// TIA Portal project "MetalCuttingLine" (V17)
// End to End

(* hardware
DEVICE "S7-1500/ET200MP station_1"  S7-1500 station
   slot 0: "Rail_0"  Rack  6ES7 590-1***0-0AA0
   slot 1: "PLC_1"  CPU 1516-3 PN/DP  6ES7 516-3AN02-0AB0  V2.9
      slot 3: "CPU display_1"  6ES7591-1BA00-0AA0
      slot 32768: "PROFINET interface_1"  X1
         slot 32769: "Port_1"  X1 P1
         slot 32770: "Port_2"  X1 P2
      slot 33024: "PROFINET interface_2"  X2
         slot 33025: "Port_1"  X2 P1
      slot 33280: "DP interface_1"  X3
      slot 34817: "Virtual CP interface port_1"  Virtual CP interface port  Virtual CP interface port
DEVICE "HMI_1"  KTP900 Basic PN
   slot 0: "HMI_1"  KTP900 Basic PN  6AV2 123-2JB03-0AX0  17.0.0.0
   slot 1: "HMI_RT_1"  KTP900 Basic PN  6AV2 123-2JB03-0AX0  17.0.0.0
   slot 5: "HMI_1.IE_CP_1"  PROFINET Interface  17.0.0.0
      slot 1: "PROFINET Interface_1"  PROFINET Interface
         slot 1: "Port_1"  Port
*)

// ===== PLC "PLC_1"  CPU 1516-3 PN/DP =====

VAR_GLOBAL   // PLC tag table "IO_Tags"
   "I_StartPB" AT %I0.0 : Bool;   // Start pushbutton
   "I_StopPB" AT %I0.1 : Bool;   // Stop pushbutton
   "I_EStop" AT %I0.2 : Bool;   // Emergency stop (NC contact)
   "I_AutoManSwitch" AT %I0.3 : Bool;   // Mode select switch
   "I_ClampRetracted" AT %I0.4 : Bool;   // Clamp cylinder retracted limit switch
   "I_ClampExtended" AT %I0.5 : Bool;   // Clamp cylinder extended limit switch
   "I_ShearRetracted" AT %I0.6 : Bool;   // Shear cylinder retracted limit switch
   "I_ShearExtended" AT %I0.7 : Bool;   // Shear cylinder extended limit switch
   "I_PartAtEject" AT %I1.0 : Bool;   // Photoeye at eject station
   "Q_FeedMotor" AT %Q0.0 : Bool;   // Feed conveyor motor run
   "Q_ClampExtend" AT %Q0.1 : Bool;   // Clamp cylinder extend solenoid
   "Q_ClampRetract" AT %Q0.2 : Bool;   // Clamp cylinder retract solenoid
   "Q_ShearExtend" AT %Q0.3 : Bool;   // Shear cylinder extend solenoid
   "Q_ShearRetract" AT %Q0.4 : Bool;   // Shear cylinder retract solenoid
   "Q_EjectGoodLane" AT %Q0.5 : Bool;   // Diverter to good-parts lane
   "Q_EjectScrapLane" AT %Q0.6 : Bool;   // Diverter to scrap lane
   "Q_RunLamp" AT %Q0.7 : Bool;   // Auto-run indicator lamp
   "Q_FaultLamp" AT %Q1.0 : Bool;   // Fault/alarm indicator lamp
END_VAR

DATA_BLOCK "Recipe_Status"   // DB1
{ S7_Optimized_Access := 'FALSE' }
VERSION : 0.1
   VAR
      Recipe : Struct
         TargetLength : Real := 500.0;   // Target cut length in mm
         Tolerance : Real := 2.0;   // Allowed+- tolerance in mm
         FeedSpeed : Real := 50.0;   // Feed Conveyor speed referenc %
      END_STRUCT;
      Status : Struct
         CurrentLength : Real := 0.0;   // Live measured length from the encoder
         GoodCount : Int;   // Total good pieces cut
         ScrapCount : Int;   // Total scrap pieces out
         TotalCount : Int;   // Total pieces cut (good+scrap)
      END_STRUCT;
      Mode : Struct
         AutoMode : Bool;   // True when in Auto mode
         ManualMode : Bool;   // True when in Manual mode
         Running : Bool;   // True when machine cycle is active
      END_STRUCT;
      Alarms : Struct
         EstopTripped : Bool;   // Emergency stop active
         ClampFault : Bool;   // Clamp cylinder failed to reach position
         ShearFault : Bool;   // Shear cylinder failed to reach position
         LengthError : Bool;   // Measured length out of expected range
         AnyFaultActive : Bool;   // True if any single fault active
         AlarmWord : Word;   // alarmWord
      END_STRUCT;
   END_VAR
BEGIN
END_DATA_BLOCK

DATA_BLOCK "ModeControl_DB"   // DB2
{ S7_Optimized_Access := 'TRUE' }
VERSION : 0.1
// stored: InstanceOfName ModeControl
"ModeControl"
BEGIN
END_DATA_BLOCK

DATA_BLOCK "FeedConveyor_DB"   // DB3
{ S7_Optimized_Access := 'TRUE' }
VERSION : 0.1
// stored: InstanceOfName FeedConveyor
"FeedConveyor"
BEGIN
END_DATA_BLOCK

DATA_BLOCK "LengthMeasurement_DB"   // DB4
{ S7_Optimized_Access := 'TRUE' }
VERSION : 0.1
// stored: InstanceOfName LengthMeasurement
"LengthMeasurement"
BEGIN
END_DATA_BLOCK

DATA_BLOCK "ShearCylinder_DB"   // DB5
{ S7_Optimized_Access := 'TRUE' }
VERSION : 0.1
// stored: InstanceOfName ShearCylinder
"ShearCylinder"
BEGIN
END_DATA_BLOCK

DATA_BLOCK "ClampCylinder_DB"   // DB6
{ S7_Optimized_Access := 'TRUE' }
VERSION : 0.1
// stored: InstanceOfName ClampCylinder
"ClampCylinder"
BEGIN
END_DATA_BLOCK

DATA_BLOCK "EjectSort_DB"   // DB7
{ S7_Optimized_Access := 'TRUE' }
VERSION : 0.1
// stored: InstanceOfName EjectSort
"EjectSort"
BEGIN
END_DATA_BLOCK

DATA_BLOCK "AlarmHandler_DB"   // DB8
{ S7_Optimized_Access := 'TRUE' }
VERSION : 0.1
// stored: InstanceOfName AlarmHandler
"AlarmHandler"
BEGIN
END_DATA_BLOCK

FUNCTION_BLOCK "ModeControl"   // FB1, LAD
{ S7_Optimized_Access := 'TRUE' }
VERSION : 0.1
   VAR_INPUT
      StartPB : Bool;
      StopPB : Bool;
      EStop : Bool;
      AutManSwitch : Bool;
   END_VAR
BEGIN

REGION Network 1: Start/Stop seal in Rung
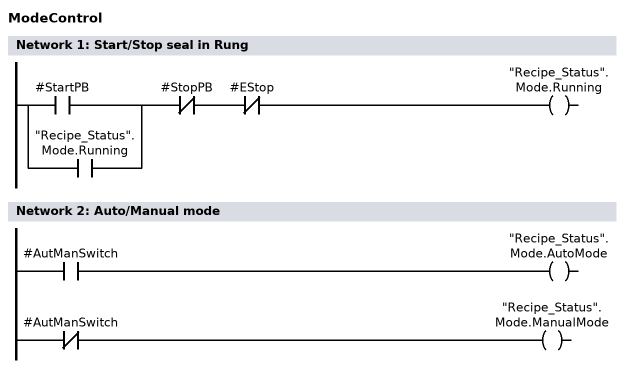
   RUNG wire#powerrail
      Contact( #StartPB )
      wire#w1
      I_Contact( #StopPB )
      I_Contact( #EStop )
      Coil( "Recipe_Status".Mode.Running )
   END_RUNG
   RUNG wire#powerrail
      Contact( "Recipe_Status".Mode.Running )
   END_RUNG wire#w1
   // the same network as SCL:
   "Recipe_Status".Mode.Running := (#StartPB OR "Recipe_Status".Mode.Running) AND NOT #StopPB AND NOT #EStop;
END_REGION

REGION Network 2: Auto/Manual mode
   RUNG wire#powerrail
      Contact( #AutManSwitch )
      Coil( "Recipe_Status".Mode.AutoMode )
   END_RUNG
   RUNG wire#powerrail
      I_Contact( #AutManSwitch )
      Coil( "Recipe_Status".Mode.ManualMode )
   END_RUNG
   // the same network as SCL:
   "Recipe_Status".Mode.AutoMode := #AutManSwitch;
   "Recipe_Status".Mode.ManualMode := NOT #AutManSwitch;
END_REGION
END_FUNCTION_BLOCK

FUNCTION_BLOCK "FeedConveyor"   // FB2, LAD
{ S7_Optimized_Access := 'TRUE' }
VERSION : 0.1
   VAR_INPUT
      LengthReached : Bool;
   END_VAR
   VAR_IN_OUT
      FeedMotorOn : Bool;
   END_VAR
BEGIN

REGION Network 1
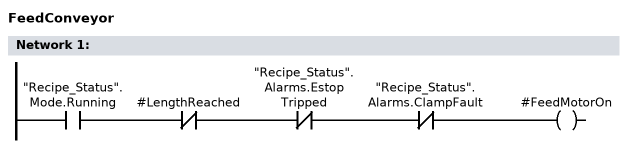
   RUNG wire#powerrail
      Contact( "Recipe_Status".Mode.Running )
      I_Contact( #LengthReached )
      I_Contact( "Recipe_Status".Alarms.EstopTripped )
      I_Contact( "Recipe_Status".Alarms.ClampFault )
      Coil( #FeedMotorOn )
   END_RUNG
   // the same network as SCL:
   #FeedMotorOn := "Recipe_Status".Mode.Running AND NOT #LengthReached AND NOT "Recipe_Status".Alarms.EstopTripped AND NOT "Recipe_Status".Alarms.ClampFault;
END_REGION
END_FUNCTION_BLOCK

FUNCTION_BLOCK "LengthMeasurement"   // FB3, LAD
{ S7_Optimized_Access := 'TRUE' }
VERSION : 0.1
   VAR_INPUT
      FeedMotorOn : Bool;
      ResetRamp : Bool;
   END_VAR
   VAR_OUTPUT
      LengthReached : Bool;
   END_VAR
   VAR
      RampAccum : Real;
      ToleranceCheck : Real;
   END_VAR
BEGIN

REGION Network 1: Accumulate Simulated Length
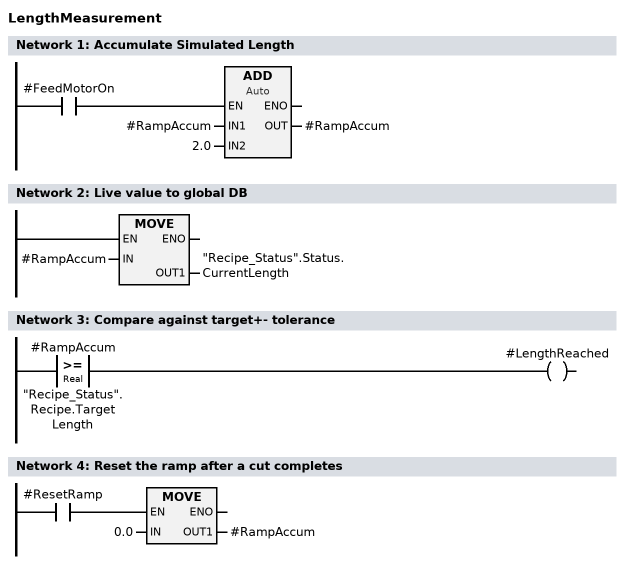
   RUNG wire#powerrail
      Contact( #FeedMotorOn )
      Add(in1 := #RampAccum, in2 := 2.0, out => #RampAccum)
   END_RUNG
   // the same network as SCL:
   IF #FeedMotorOn THEN #RampAccum := #RampAccum + 2.0; END_IF;
END_REGION

REGION Network 2: Live value to global DB
   RUNG wire#powerrail
      Move(in := #RampAccum, out1 => "Recipe_Status".Status.CurrentLength)
   END_RUNG
   // the same network as SCL:
   "Recipe_Status".Status.CurrentLength := #RampAccum;
END_REGION

REGION Network 3: Compare against target+- tolerance
   RUNG wire#powerrail
      { S7_Templates := "SrcType := Real" } GE_Contact(in1 := #RampAccum, in2 := "Recipe_Status".Recipe.TargetLength)
      Coil( #LengthReached )
   END_RUNG
   // the same network as SCL:
   #LengthReached := #RampAccum >= "Recipe_Status".Recipe.TargetLength;
END_REGION

REGION Network 4: Reset the ramp after a cut completes
   RUNG wire#powerrail
      Contact( #ResetRamp )
      Move(in := 0.0, out1 => #RampAccum)
   END_RUNG
   // the same network as SCL:
   IF #ResetRamp THEN #RampAccum := 0.0; END_IF;
END_REGION
END_FUNCTION_BLOCK

FUNCTION_BLOCK "ClampCylinder"   // FB4, LAD
{ S7_Optimized_Access := 'TRUE' }
VERSION : 0.1
   VAR_INPUT
      StartClamp : Bool;
      RetractClamp : Bool;
      ClampRetractedSensor : Bool;
      ClampExtendedSensor : Bool;
   END_VAR
   VAR_OUTPUT
      ClampExtendedCoil : Bool;
      ClampRetractCoil : Bool;
      ClampInPosition : Bool;
   END_VAR
   VAR
      "Step" : Int;
   END_VAR
   VAR_TEMP   // added for the SCL form of the ladder/FBD networks
      _w1 : Bool;
   END_VAR
BEGIN

REGION Network 1: Step0--> Step1 (Start Extending)
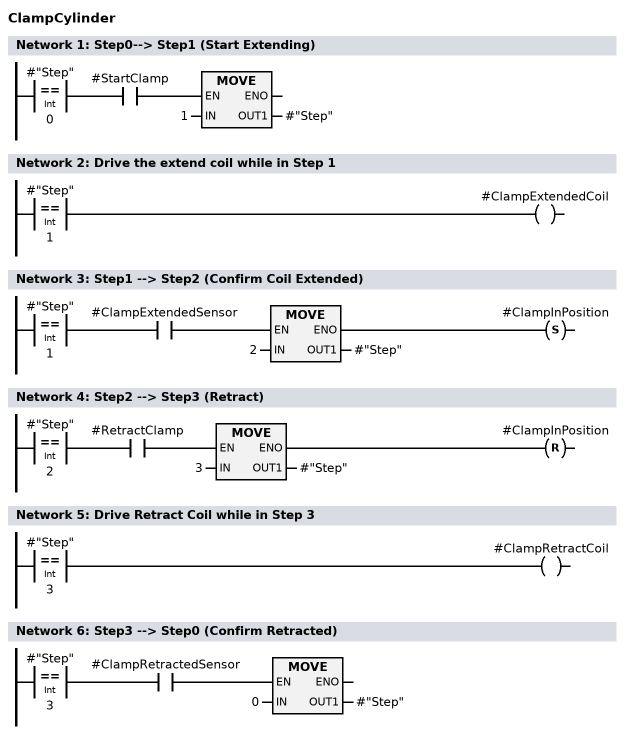
   RUNG wire#powerrail
      { S7_Templates := "SrcType := Int" } EQ_Contact(in1 := #"Step", in2 := 0)
      Contact( #StartClamp )
      Move(in := 1, out1 => #"Step")
   END_RUNG
   // the same network as SCL:
   IF (#"Step" = 0) AND #StartClamp THEN #"Step" := 1; END_IF;
END_REGION

REGION Network 2: Drive the extend coil while in Step 1
   RUNG wire#powerrail
      { S7_Templates := "SrcType := Int" } EQ_Contact(in1 := #"Step", in2 := 1)
      Coil( #ClampExtendedCoil )
   END_RUNG
   // the same network as SCL:
   #ClampExtendedCoil := #"Step" = 1;
END_REGION

REGION Network 3: Step1 --> Step2 (Confirm Coil Extended)
   RUNG wire#powerrail
      { S7_Templates := "SrcType := Int" } EQ_Contact(in1 := #"Step", in2 := 1)
      Contact( #ClampExtendedSensor )
      Move(in := 2, out1 => #"Step")
      S_Coil( #ClampInPosition )
   END_RUNG
   // the same network as SCL:
   #_w1 := (#"Step" = 1) AND #ClampExtendedSensor;
   IF #_w1 THEN
       #"Step" := 2;
       #ClampInPosition := TRUE;
   END_IF;
END_REGION

REGION Network 4: Step2 --> Step3 (Retract)
   RUNG wire#powerrail
      { S7_Templates := "SrcType := Int" } EQ_Contact(in1 := #"Step", in2 := 2)
      Contact( #RetractClamp )
      Move(in := 3, out1 => #"Step")
      R_Coil( #ClampInPosition )
   END_RUNG
   // the same network as SCL:
   #_w1 := (#"Step" = 2) AND #RetractClamp;
   IF #_w1 THEN
       #"Step" := 3;
       #ClampInPosition := FALSE;
   END_IF;
END_REGION

REGION Network 5: Drive Retract Coil while in Step 3
   RUNG wire#powerrail
      { S7_Templates := "SrcType := Int" } EQ_Contact(in1 := #"Step", in2 := 3)
      Coil( #ClampRetractCoil )
   END_RUNG
   // the same network as SCL:
   #ClampRetractCoil := #"Step" = 3;
END_REGION

REGION Network 6: Step3 --> Step0 (Confirm Retracted)
   RUNG wire#powerrail
      { S7_Templates := "SrcType := Int" } EQ_Contact(in1 := #"Step", in2 := 3)
      Contact( #ClampRetractedSensor )
      Move(in := 0, out1 => #"Step")
   END_RUNG
   // the same network as SCL:
   IF (#"Step" = 3) AND #ClampRetractedSensor THEN #"Step" := 0; END_IF;
END_REGION
END_FUNCTION_BLOCK

FUNCTION_BLOCK "ShearCylinder"   // FB5, LAD
{ S7_Optimized_Access := 'TRUE' }
VERSION : 0.1
   VAR_INPUT
      StartShear : Bool;
      ShearRetractedSensor : Bool;
      ShearExtendedSensor : Bool;
   END_VAR
   VAR_OUTPUT
      ShearExtendCoil : Bool;
      ShearRetractCoil : Bool;
      CutComplete : Bool;
   END_VAR
   VAR
      "Step" : Int;
      FaultTimer : IEC_TIMER;
   END_VAR
   VAR_TEMP   // added for the SCL form of the ladder/FBD networks
      _w1 : Bool;
   END_VAR
BEGIN

REGION Network 1: Start Extending
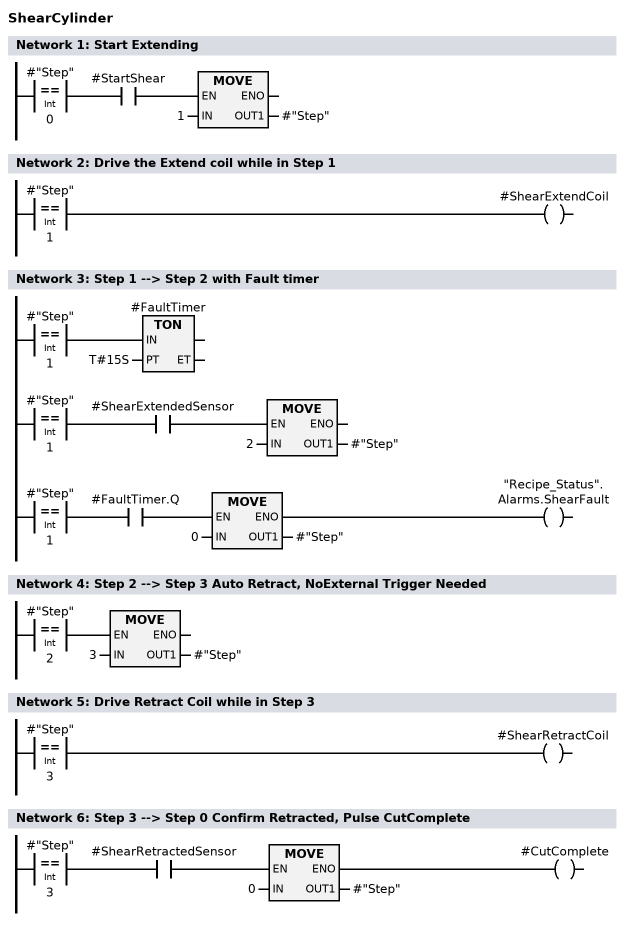
   RUNG wire#powerrail
      { S7_Templates := "SrcType := Int" } EQ_Contact(in1 := #"Step", in2 := 0)
      Contact( #StartShear )
      Move(in := 1, out1 => #"Step")
   END_RUNG
   // the same network as SCL:
   IF (#"Step" = 0) AND #StartShear THEN #"Step" := 1; END_IF;
END_REGION

REGION Network 2: Drive the Extend coil while in Step 1
   RUNG wire#powerrail
      { S7_Templates := "SrcType := Int" } EQ_Contact(in1 := #"Step", in2 := 1)
      Coil( #ShearExtendCoil )
   END_RUNG
   // the same network as SCL:
   #ShearExtendCoil := #"Step" = 1;
END_REGION

REGION Network 3: Step 1 --> Step 2 with Fault timer
   #FaultTimer.TON(IN := #"Step" = 1, PT := T#15S);
   IF (#"Step" = 1) AND #ShearExtendedSensor THEN #"Step" := 2; END_IF;
   #_w1 := (#"Step" = 1) AND #FaultTimer.Q;
   IF #_w1 THEN #"Step" := 0; END_IF;
   "Recipe_Status".Alarms.ShearFault := #_w1;
END_REGION

REGION Network 4: Step 2 --> Step 3 Auto Retract, NoExternal Trigger Needed
   RUNG wire#powerrail
      { S7_Templates := "SrcType := Int" } EQ_Contact(in1 := #"Step", in2 := 2)
      Move(in := 3, out1 => #"Step")
   END_RUNG
   // the same network as SCL:
   IF #"Step" = 2 THEN #"Step" := 3; END_IF;
END_REGION

REGION Network 5: Drive Retract Coil while in Step 3
   RUNG wire#powerrail
      { S7_Templates := "SrcType := Int" } EQ_Contact(in1 := #"Step", in2 := 3)
      Coil( #ShearRetractCoil )
   END_RUNG
   // the same network as SCL:
   #ShearRetractCoil := #"Step" = 3;
END_REGION

REGION Network 6: Step 3 --> Step 0 Confirm Retracted, Pulse CutComplete
   RUNG wire#powerrail
      { S7_Templates := "SrcType := Int" } EQ_Contact(in1 := #"Step", in2 := 3)
      Contact( #ShearRetractedSensor )
      Move(in := 0, out1 => #"Step")
      Coil( #CutComplete )
   END_RUNG
   // the same network as SCL:
   #_w1 := (#"Step" = 3) AND #ShearRetractedSensor;
   IF #_w1 THEN #"Step" := 0; END_IF;
   #CutComplete := #_w1;
END_REGION
END_FUNCTION_BLOCK

FUNCTION_BLOCK "EjectSort"   // FB6, LAD
{ S7_Optimized_Access := 'TRUE' }
VERSION : 0.1
   VAR_INPUT
      PartAtEject : Bool;
   END_VAR
   VAR_OUTPUT
      EjectGoodCoil : Bool;
      EjectScrapCoil : Bool;
   END_VAR
   VAR
      GoodEdgeMem : Bool;
      ScrapEdgeMem : Bool;
   END_VAR
   VAR_TEMP
      LengthDiff : Real;
      WithinTolerance : Bool;
   END_VAR
   VAR_TEMP   // added for the SCL form of the ladder/FBD networks
      _w1 : Bool;
      _w2 : Bool;
   END_VAR
BEGIN

REGION Network 1: Calculate whether the cut was within tolerance
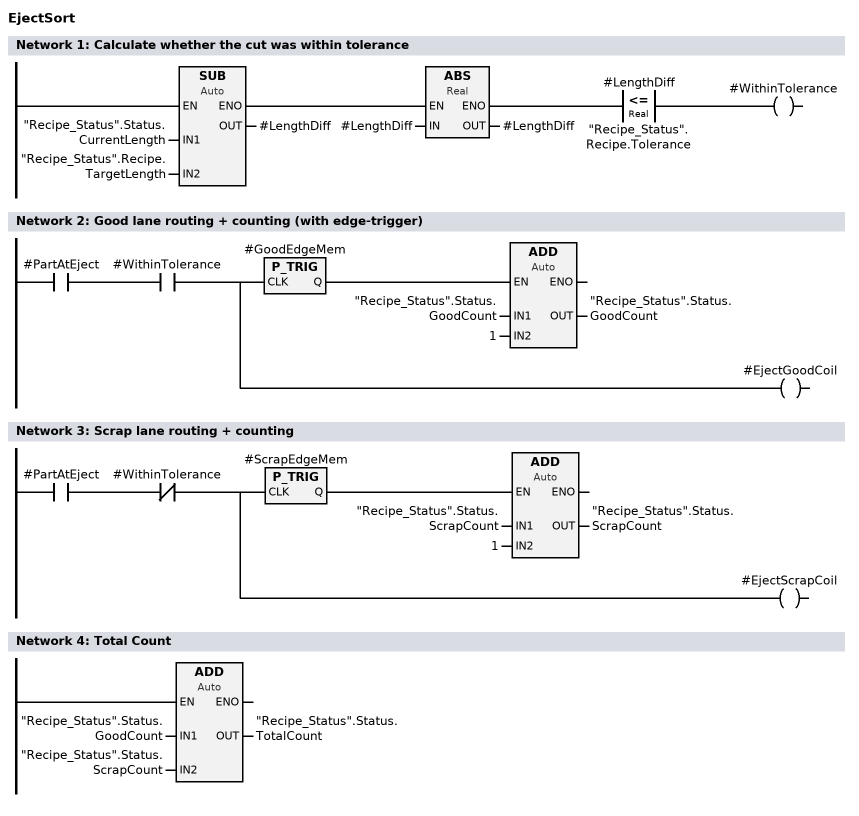
   RUNG wire#powerrail
      Sub(in1 := "Recipe_Status".Status.CurrentLength, in2 := "Recipe_Status".Recipe.TargetLength, out => #LengthDiff)
      { S7_Templates := "SrcType := Real" } Abs(in := #LengthDiff, out => #LengthDiff)
      { S7_Templates := "SrcType := Real" } LE_Contact(in1 := #LengthDiff, in2 := "Recipe_Status".Recipe.Tolerance)
      Coil( #WithinTolerance )
   END_RUNG
   // the same network as SCL:
   #LengthDiff := "Recipe_Status".Status.CurrentLength - "Recipe_Status".Recipe.TargetLength;
   #LengthDiff := ABS(#LengthDiff);
   #WithinTolerance := #LengthDiff <= "Recipe_Status".Recipe.Tolerance;
END_REGION

REGION Network 2: Good lane routing + counting (with edge-trigger)
   RUNG wire#powerrail
      Contact( #PartAtEject )
      Contact( #WithinTolerance )
      wire#w1
      P_Trig( #GoodEdgeMem )
      Add(in1 := "Recipe_Status".Status.GoodCount, in2 := 1, out => "Recipe_Status".Status.GoodCount)
   END_RUNG
   RUNG wire#w1
      Coil( #EjectGoodCoil )
   END_RUNG
   // the same network as SCL:
   #_w1 := #PartAtEject AND #WithinTolerance;
   #_w2 := #_w1 AND NOT #GoodEdgeMem;   // rising edge
   #GoodEdgeMem := #_w1;
   IF #_w2 THEN "Recipe_Status".Status.GoodCount := "Recipe_Status".Status.GoodCount + 1; END_IF;
   #EjectGoodCoil := #_w1;
END_REGION

REGION Network 3: Scrap lane routing + counting
   RUNG wire#powerrail
      Contact( #PartAtEject )
      I_Contact( #WithinTolerance )
      wire#w1
      P_Trig( #ScrapEdgeMem )
      Add(in1 := "Recipe_Status".Status.ScrapCount, in2 := 1, out => "Recipe_Status".Status.ScrapCount)
   END_RUNG
   RUNG wire#w1
      Coil( #EjectScrapCoil )
   END_RUNG
   // the same network as SCL:
   #_w1 := #PartAtEject AND NOT #WithinTolerance;
   #_w2 := #_w1 AND NOT #ScrapEdgeMem;   // rising edge
   #ScrapEdgeMem := #_w1;
   IF #_w2 THEN "Recipe_Status".Status.ScrapCount := "Recipe_Status".Status.ScrapCount + 1; END_IF;
   #EjectScrapCoil := #_w1;
END_REGION

REGION Network 4: Total Count
   RUNG wire#powerrail
      Add(in1 := "Recipe_Status".Status.GoodCount, in2 := "Recipe_Status".Status.ScrapCount, out => "Recipe_Status".Status.TotalCount)
   END_RUNG
   // the same network as SCL:
   "Recipe_Status".Status.TotalCount := "Recipe_Status".Status.GoodCount + "Recipe_Status".Status.ScrapCount;
END_REGION
END_FUNCTION_BLOCK

FUNCTION_BLOCK "AlarmHandler"   // FB7, LAD
{ S7_Optimized_Access := 'TRUE' }
VERSION : 0.1
BEGIN

REGION Network 1: Combine all faults into one bit
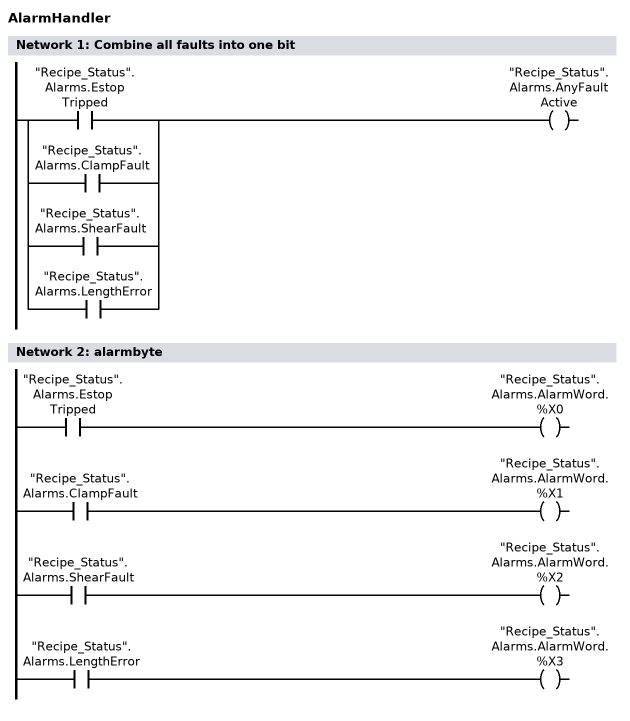
   RUNG wire#powerrail
      Contact( "Recipe_Status".Alarms.EstopTripped )
      wire#w1
      Coil( "Recipe_Status".Alarms.AnyFaultActive )
   END_RUNG
   RUNG wire#powerrail
      Contact( "Recipe_Status".Alarms.ClampFault )
   END_RUNG wire#w1
   RUNG wire#powerrail
      Contact( "Recipe_Status".Alarms.ShearFault )
   END_RUNG wire#w1
   RUNG wire#powerrail
      Contact( "Recipe_Status".Alarms.LengthError )
   END_RUNG wire#w1
   // the same network as SCL:
   "Recipe_Status".Alarms.AnyFaultActive := "Recipe_Status".Alarms.EstopTripped OR "Recipe_Status".Alarms.ClampFault OR "Recipe_Status".Alarms.ShearFault OR "Recipe_Status".Alarms.LengthError;
END_REGION

REGION Network 2: alarmbyte
   RUNG wire#powerrail
      Contact( "Recipe_Status".Alarms.EstopTripped )
      Coil( "Recipe_Status".Alarms.AlarmWord.%X0 )
   END_RUNG
   RUNG wire#powerrail
      Contact( "Recipe_Status".Alarms.ClampFault )
      Coil( "Recipe_Status".Alarms.AlarmWord.%X1 )
   END_RUNG
   RUNG wire#powerrail
      Contact( "Recipe_Status".Alarms.ShearFault )
      Coil( "Recipe_Status".Alarms.AlarmWord.%X2 )
   END_RUNG
   RUNG wire#powerrail
      Contact( "Recipe_Status".Alarms.LengthError )
      Coil( "Recipe_Status".Alarms.AlarmWord.%X3 )
   END_RUNG
   // the same network as SCL:
   "Recipe_Status".Alarms.AlarmWord.%X0 := "Recipe_Status".Alarms.EstopTripped;
   "Recipe_Status".Alarms.AlarmWord.%X1 := "Recipe_Status".Alarms.ClampFault;
   "Recipe_Status".Alarms.AlarmWord.%X2 := "Recipe_Status".Alarms.ShearFault;
   "Recipe_Status".Alarms.AlarmWord.%X3 := "Recipe_Status".Alarms.LengthError;
END_REGION
END_FUNCTION_BLOCK

ORGANIZATION_BLOCK "Main"   // OB1, LAD, ProgramCycle
TITLE = "Main Program Sweep (Cycle)"
{ S7_Optimized_Access := 'TRUE' }
VERSION : 0.1
   VAR_INPUT
      Initial_Call : Bool;   // Initial call of this OB
      Remanence : Bool;   // =True, if remanent data are available
   END_VAR
BEGIN

REGION Network 1
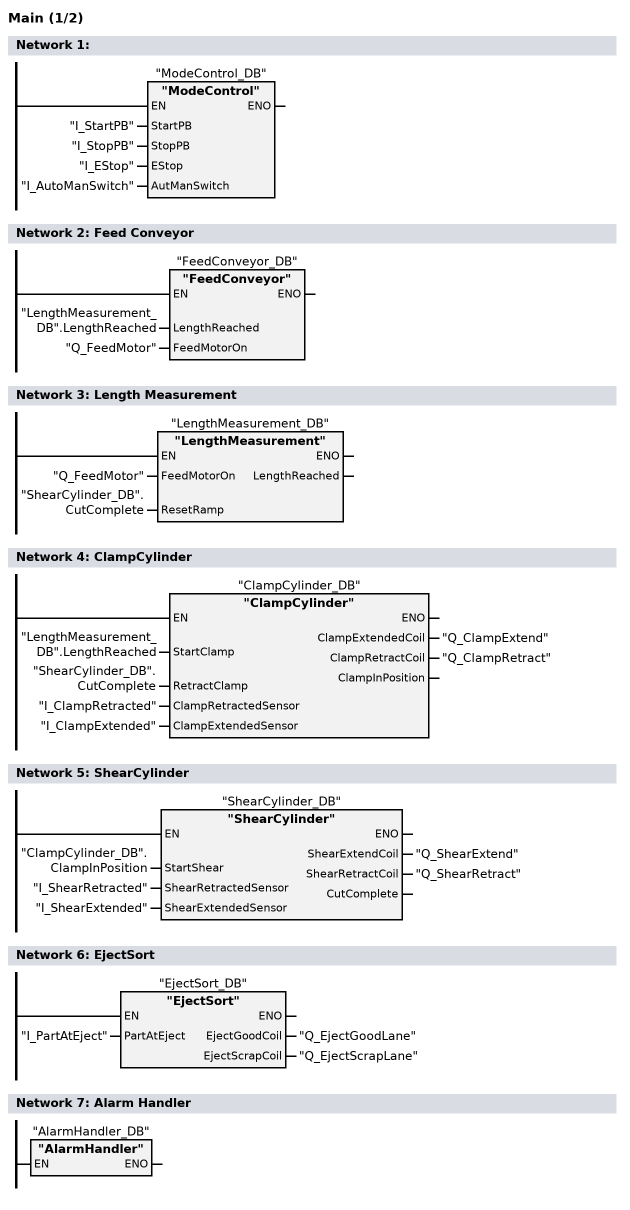
   RUNG wire#powerrail
      "ModeControl_DB"(StartPB := "I_StartPB", StopPB := "I_StopPB", EStop := "I_EStop", AutManSwitch := "I_AutoManSwitch")
   END_RUNG
   // the same network as SCL:
   "ModeControl_DB"(StartPB := "I_StartPB",   // "ModeControl"
                    StopPB := "I_StopPB",
                    EStop := "I_EStop",
                    AutManSwitch := "I_AutoManSwitch");
END_REGION

REGION Network 2: Feed Conveyor
   RUNG wire#powerrail
      "FeedConveyor_DB"(LengthReached := "LengthMeasurement_DB".LengthReached, FeedMotorOn := "Q_FeedMotor")
   END_RUNG
   // the same network as SCL:
   "FeedConveyor_DB"(LengthReached := "LengthMeasurement_DB".LengthReached, FeedMotorOn := "Q_FeedMotor");   // "FeedConveyor"
END_REGION

REGION Network 3: Length Measurement
   RUNG wire#powerrail
      "LengthMeasurement_DB"(FeedMotorOn := "Q_FeedMotor", ResetRamp := "ShearCylinder_DB".CutComplete, LengthReached =>)
   END_RUNG
   // the same network as SCL:
   "LengthMeasurement_DB"(FeedMotorOn := "Q_FeedMotor", ResetRamp := "ShearCylinder_DB".CutComplete);   // "LengthMeasurement"
END_REGION

REGION Network 4: ClampCylinder
   RUNG wire#powerrail
      "ClampCylinder_DB"(StartClamp := "LengthMeasurement_DB".LengthReached, RetractClamp := "ShearCylinder_DB".CutComplete, ClampRetractedSensor := "I_ClampRetracted", ClampExtendedSensor := "I_ClampExtended", ClampExtendedCoil => "Q_ClampExtend", ClampRetractCoil => "Q_ClampRetract", ClampInPosition =>)
   END_RUNG
   // the same network as SCL:
   "ClampCylinder_DB"(StartClamp := "LengthMeasurement_DB".LengthReached,   // "ClampCylinder"
                      RetractClamp := "ShearCylinder_DB".CutComplete,
                      ClampRetractedSensor := "I_ClampRetracted",
                      ClampExtendedSensor := "I_ClampExtended",
                      ClampExtendedCoil => "Q_ClampExtend",
                      ClampRetractCoil => "Q_ClampRetract");
END_REGION

REGION Network 5: ShearCylinder
   RUNG wire#powerrail
      "ShearCylinder_DB"(StartShear := "ClampCylinder_DB".ClampInPosition, ShearRetractedSensor := "I_ShearRetracted", ShearExtendedSensor := "I_ShearExtended", ShearExtendCoil => "Q_ShearExtend", ShearRetractCoil => "Q_ShearRetract", CutComplete =>)
   END_RUNG
   // the same network as SCL:
   "ShearCylinder_DB"(StartShear := "ClampCylinder_DB".ClampInPosition,   // "ShearCylinder"
                      ShearRetractedSensor := "I_ShearRetracted",
                      ShearExtendedSensor := "I_ShearExtended",
                      ShearExtendCoil => "Q_ShearExtend",
                      ShearRetractCoil => "Q_ShearRetract");
END_REGION

REGION Network 6: EjectSort
   RUNG wire#powerrail
      "EjectSort_DB"(PartAtEject := "I_PartAtEject", EjectGoodCoil => "Q_EjectGoodLane", EjectScrapCoil => "Q_EjectScrapLane")
   END_RUNG
   // the same network as SCL:
   "EjectSort_DB"(PartAtEject := "I_PartAtEject",   // "EjectSort"
                  EjectGoodCoil => "Q_EjectGoodLane",
                  EjectScrapCoil => "Q_EjectScrapLane");
END_REGION

REGION Network 7: Alarm Handler
   RUNG wire#powerrail
      "AlarmHandler_DB"()
   END_RUNG
   // the same network as SCL:
   "AlarmHandler_DB"();   // "AlarmHandler"
END_REGION

REGION Network 8: Run/ Fault Lmaps
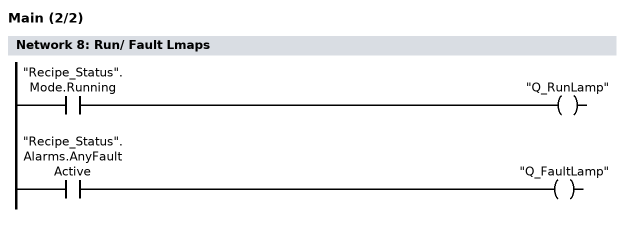
   RUNG wire#powerrail
      Contact( "Recipe_Status".Mode.Running )
      Coil( "Q_RunLamp" )
   END_RUNG
   RUNG wire#powerrail
      Contact( "Recipe_Status".Alarms.AnyFaultActive )
      Coil( "Q_FaultLamp" )
   END_RUNG
   // the same network as SCL:
   "Q_RunLamp" := "Recipe_Status".Mode.Running;
   "Q_FaultLamp" := "Recipe_Status".Alarms.AnyFaultActive;
END_REGION
END_ORGANIZATION_BLOCK

(* ===== HMI "HMI_RT_1" =====
system functions are stored by id; their names below are inferred from use
connection "HMI_Connection_1": ETHERNET, SMART_S7_1500_OMS

HMI tags "Default tag table"
   "Tag_ScreenNumber" : UInt, internal
   "Q_FeedMotor" : Bool = PLC Q_FeedMotor AT %Q0.0, 1 s
   "ClampCylinder_DB_ClampInPosition" : Bool = PLC ClampCylinder_DB.ClampInPosition, 1 s
   "Q_ShearExtend" : Bool = PLC Q_ShearExtend AT %Q0.3, 1 s
   "I_PartAtEject" : Bool = PLC I_PartAtEject AT %I1.0, 1 s
   "I_StartPB" : Bool = PLC I_StartPB AT %I0.0, 1 s
   "I_StopPB" : Bool = PLC I_StopPB AT %I0.1, 1 s
   "Recipe_Status_Mode_Running" : Bool = PLC Recipe_Status.Mode.Running AT %DB1.DBX22.2, 1 s
   "Recipe_Status_Alarms_AnyFaultActive" : Bool = PLC Recipe_Status.Alarms.AnyFaultActive AT %DB1.DBX24.4, 1 s
   "Recipe_Status_Recipe_TargetLength" : Real = PLC Recipe_Status.Recipe.TargetLength AT %DB1.DBD0, 1 s
   "Recipe_Status_Recipe_Tolerance" : Real = PLC Recipe_Status.Recipe.Tolerance AT %DB1.DBD4, 1 s
   "Recipe_Status_Recipe_FeedSpeed" : Real = PLC Recipe_Status.Recipe.FeedSpeed AT %DB1.DBD8, 1 s
   "Recipe_Status_Alarms_EstopTripped" : Bool = PLC Recipe_Status.Alarms.EstopTripped AT %DB1.DBX24.0, 1 s
   "Recipe_Status_Alarms_ClampFault" : Bool = PLC Recipe_Status.Alarms.ClampFault AT %DB1.DBX24.1, 1 s
   "Recipe_Status_Alarms_ShearFault" : Bool = PLC Recipe_Status.Alarms.ShearFault AT %DB1.DBX24.2, 1 s
   "Recipe_Status_Alarms_LengthError" : Bool = PLC Recipe_Status.Alarms.LengthError AT %DB1.DBX24.3, 1 s
   "ShearCylinder_DB_Step" : Int = PLC ShearCylinder_DB.Step, 1 s
   "FeedConveyor_DB_FeedMotorOn" : Bool = PLC FeedConveyor_DB.FeedMotorOn, 1 s
   "Recipe_Status_Status_GoodCount" : Int = PLC Recipe_Status.Status.GoodCount AT %DB1.DBW16, 1 s
   "AlarmWord" : Word = PLC Recipe_Status.Alarms.AlarmWord AT %DB1.DBW26, 1 s
   "Recipe_Status_Status_CurrentLength" : Real = PLC Recipe_Status.Status.CurrentLength AT %DB1.DBD12, 1 s

discrete alarms
   1: 'Emergency Stop Tripped', class Errors, trigger "AlarmWord" bit 0
   2: 'Clamp Cylinder Fault', class Errors, trigger "AlarmWord" bit 1
   4: 'Shear Cylinder Fault', class Errors, trigger "AlarmWord" bit 3
   3: 'Shear Cylinder Fault', class Errors, trigger "AlarmWord" bit 2

Template "Template_1" 800x480
   Button "Exit" at 722,440 size 55x39; TextOff 'Exit'; PictureOff "ExitRuntime_KTP900_Basic_PN_TR"; PictureOn "ExitRuntime_KTP900_Basic_PN_TR"
      on Release: StopRuntime(0)
   Button "Template_Button" at 622,440 size 55x39; TextOff 'Text'
   Button "Template_Button_1" at 522,440 size 55x39; TextOff 'Text'
   Button "Template_Button_2" at 422,440 size 55x39; TextOff 'Text'
   Button "Template_Button_3" at 322,440 size 55x39; TextOff 'Text'
   Button "Template_Button_4" at 222,440 size 55x39; TextOff 'Text'
   Button "Alarms" at 122,440 size 55x39; TextOff 'Alarms'; PictureOff "AlarmDisplay_KTP900_Basic_PN_TR"; PictureOn "AlarmDisplay_KTP900_Basic_PN_TR"
      on Release: function_ef3f5d25("Alarm window_Unacknowledged", -1)
   Button "Start screen" at 22,440 size 55x39; TextOff 'Start screen'; PictureOff "NavigateHome_KTP900_Basic_PN_TR"; PictureOn "NavigateHome_KTP900_Basic_PN_TR"
      on Release: ActivateScreen("Overview", 0)
   SymbolicIOField "Symbolic_IO_Field_Screen" at 73,7 size 620x26; TextOff '0'; TextOn '1'; TextList "TextList_ScreenNames"
      ProcessValue <- "Tag_ScreenNumber"
      on Change: ActivateScreenByNumber("Tag_ScreenNumber", 0)
   DateTimeField "HmiScreenItemData" at 695,20 size 105x20
   DateTimeField "HmiScreenItemData_1" at 695,0 size 105x20
   GraphicView "Logo" at 0,0 size 71x40; Picture "Logo of HMI_1"

screen "Overview" 800x480, template "Template_1"
   on GenerateScreen: SetTag("Tag_ScreenNumber", 1)
   Rectangle "Rectangle_1" at 1,70 size 199x41
      Appearance <- "Q_FeedMotor"
   Rectangle "Rectangle_2" at 208,71 size 201x42
      Appearance <- "ClampCylinder_DB_ClampInPosition"
   Rectangle "Rectangle_3" at 417,71 size 199x42
      Appearance <- "Q_ShearExtend"
   Rectangle "Rectangle_4" at 623,71 size 168x42
      Appearance <- "I_PartAtEject"
   Button "Button_1" at 43,138 size 96x32; TextOff 'START'
      on Press: SetBit("I_StartPB")
      on Release: ResetBit("I_StartPB")
   Button "Button_2" at 688,138 size 96x32; TextOff 'STOP'
      on Press: SetBit("I_StopPB")
      on Release: ResetBit("I_StopPB")
   Circle "Circle_1" at 62,227 size 53x53
      Appearance <- "Recipe_Status_Mode_Running"
   Circle "Circle_2" at 62,317 size 54x54
      Appearance <- "Recipe_Status_Alarms_AnyFaultActive"
   Button "Button_3" at 208,229 size 113x50; TextOff 'RECIPE'
      on Click: ActivateScreen("Recipe", 0)
   Button "Button_4" at 544,230 size 113x50; TextOff 'TRENDS'
      on Click: ActivateScreen("Trends", 0)
   Button "Button_5" at 377,230 size 113x50; TextOff 'ALARMS'
      on Click: ActivateScreen("Alarms", 0)

screen "Alarms" 800x480
   AlarmView "Alarm view_1" at 5,17 size 451x115
   Button "Button_1" at 582,38 size 120x48; TextOff 'OVERVIEW'
      on Activate: ActivateScreen("Overview", 0)

screen "Recipe" 800x480
   IOField "I/O field_1" at 7,32 size 134x42; FormatPattern s999999999.999
      ProcessValue <- "Recipe_Status_Recipe_TargetLength"
   TextField "Text field_1" at 4,80 size 141x20; Text 'TARGET LENGTH (mm)'
   IOField "I/O field_2" at 180,31 size 153x42; FormatPattern s999999999.999
      ProcessValue <- "Recipe_Status_Recipe_Tolerance"
   TextField "Text field_2" at 203,79 size 115x20; Text 'TOLERANCE (mm)'
   IOField "I/O field_3" at 354,31 size 153x42; FormatPattern s999999999.999
      ProcessValue <- "Recipe_Status_Recipe_FeedSpeed"
   TextField "Text field_3" at 372,80 size 107x20; Text 'FEED SPEED (%)'
   Button "Button_1" at 580,31 size 140x44; TextOff 'OVERVIEW'
      on Click: ActivateScreen("Overview", 0)

screen "Trends" 800x480
   TrendView "Trend view_1" at 0,0 size 799x430
   Button "Button_1" at 681,442 size 96x32; TextOff 'OVERVIEW'
      on Click: ActivateScreen("Overview", 0)
*)